TYPE T_Map_Entry : ST_MAP_ENTRY; END_TYPE

(* stored: Version 1.1.0.1, ProductVersion 3.1.4024.4
   DUT T_Map_Entry: Id {9d48cdbd-c2ed-04ae-14e6-eed38472376b} *)
